Universal Robots PolyScope program: cube_dev.urp

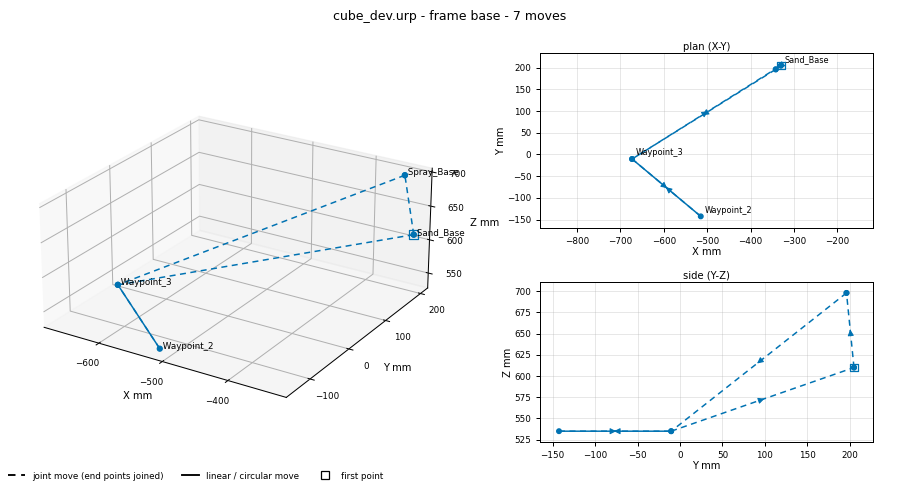
[picture p0: tool path of cube_dev.urp in frame base, 7 of 7 moves have a stored position in this frame; points joined in program order, loops and branches not executed]
Program cube_dev (installation=default directory=/programs/cube createdIn=5.11.5.1010327 lastSavedIn=5.11.5.1010327 robotSerialNumber=20215500677)
Calibrated DH parameters: a=[0.000204, -0.239222, -0.391845, -0.000001, 0.000022, 0]; d=[0.162722, -355.808559, 353.37206, 2.570385, 0.099741, 0.099629]; alpha=[1.571124, 0.000988, 0.008295, 1.568963, -1.570303, 0]; deltaTheta=[0, -0.973091, 7.204745, 0.05153, 0, 0]
Robot Program (runOnlyOnce=true)
  MoveJ speed 120 deg/s, acceleration 120 deg/s^2 (useActiveTCP=false) tcp=SandTCP; feature=Point_1
    Waypoint Sand_Base: TCP in base x=-330.026 y=205.009 z=609.986 mm, rx=0.0001 ry=-0.0003 rz=-2.2419 rad; joints [-54.6, -77.456, 120.707, 90.609, -79.088, -168.284] deg; TCP offset x=1.003 y=125.541 z=104.154 mm, rx=-0.7854 ry=0 rz=0 rad; feature pose in base x=-330 y=205 z=610 mm, rx=0 ry=0 rz=-1.5843 rad
  Folder Sand
    MoveL speed 50 mm/s, acceleration 1200 mm/s^2 (useActiveTCP=false) tcp=SandTCP; feature=Base
      MoveDirectionNode (selectedDirection=ZPlus)
        Until TOOL_CONTACT_DETECTION (allowActions=false retraction=0.001 decelerationAcceleration=3 decelerationAngularAcceleration=34.906585)
      URCap Finishing Tool Control (Robotiq_Copilot, Robotiq Inc.) dataModel(ToolOutputNameKey=SanderOn, HackTriggeringContributionIsDefinedMethodKey=true)
    MoveL speed 50 mm/s, acceleration 1200 mm/s^2 (useActiveTCP=true) feature=Base
      Force Simple feature=Base; selection=[0, 0, 1, 0, 0, 0]; wrench=[0, 0, 5, 0, 0, 0]; limitsForce=[0.15, 0.15, 0.15, 1.047198, 1.047198, 1.047198]; limitsMotion=[0.1, 0.1, 0.1, 0.349066, 0.349066, 0.349066]
        MoveDirectionNode (selectedDirection=XMinus)
          Until DISTANCE (allowActions=false deceleration=3 distanceNodeType=BLEND) Distance=0.355; motionParameters(blendRadius=0.025)
        MoveDirectionNode (selectedDirection=YMinus)
          Until DISTANCE (allowActions=false deceleration=3 distanceNodeType=BLEND) Distance=0.355; motionParameters(blendRadius=0.025)
        MoveDirectionNode (selectedDirection=XPlus)
          Until DISTANCE (allowActions=false deceleration=3 distanceNodeType=BLEND) Distance=0.355; motionParameters(blendRadius=0.025)
        MoveDirectionNode (selectedDirection=YPlus)
          Until DISTANCE (allowActions=false deceleration=3 distanceNodeType=STOP) Distance=0.355; motionParameters(blendRadius=0.01)
        URCap Finishing Tool Control (Robotiq_Copilot, Robotiq Inc.) dataModel(FinishingToolStateKey=false, ToolOutputNameKey=SanderOn, HackTriggeringContributionIsDefinedMethodKey=true)
    MoveL speed 90 mm/s, acceleration 1200 mm/s^2 (useActiveTCP=false) tcp=SandTCP; feature=Base
      MoveDirectionNode (selectedDirection=ZMinus)
        Until DISTANCE (allowActions=false deceleration=3 distanceNodeType=BLEND) Distance=0.05; motionParameters(blendRadius=0.003)
  Folder Spray Vert
    MoveJ speed 120 deg/s, acceleration 150 deg/s^2 (useActiveTCP=false) tcp=SprayTCP; feature=Point_1
      Waypoint Spray_Base: TCP in base x=-341.952 y=196.173 z=697.866 mm, rx=0 ry=0 rz=0.0032 rad; joints [-64.094, -80.171, 99.151, 94.355, -50.864, 55.964] deg; TCP offset x=-61.38 y=-97.07 z=93.78 mm, rx=0.6139 ry=0.6139 rz=-1.4822 rad; feature pose in base x=-341.965 y=196.202 z=697.85 mm, rx=0 ry=0 rz=-1.5843 rad
    MoveL speed 90 mm/s, acceleration 1200 mm/s^2 (useActiveTCP=false) tcp=SprayTCP; feature=Base
      MoveDirectionNode (selectedDirection=ZMinus)
        Until DISTANCE (allowActions=false deceleration=3 distanceNodeType=BLEND) Distance=0.05; motionParameters(blendRadius=0.003)
      Set DigitalOutput pin=SprayerOn; digitalValue=1
      MoveDirectionNode (selectedDirection=XMinus)
        Until DISTANCE (allowActions=false deceleration=3 distanceNodeType=BLEND) Distance=0.355; motionParameters(blendRadius=0.003)
      MoveDirectionNode (selectedDirection=YMinus)
        Until DISTANCE (allowActions=false deceleration=3 distanceNodeType=BLEND) Distance=0.355; motionParameters(blendRadius=0.003)
      MoveDirectionNode (selectedDirection=XPlus)
        Until DISTANCE (allowActions=false deceleration=3 distanceNodeType=BLEND) Distance=0.355; motionParameters(blendRadius=0.003)
      MoveDirectionNode (selectedDirection=YPlus)
        Until DISTANCE (allowActions=false deceleration=3 distanceNodeType=BLEND) Distance=0.355; motionParameters(blendRadius=0.003)
      Set DigitalOutput pin=SprayerOn; digitalValue=0
  Folder Spray Horiz
    MoveJ speed 120 deg/s, acceleration 150 deg/s^2 (useActiveTCP=false) tcp=SprayTCP; feature=Point_1
      Waypoint Spray_Base: TCP in base x=-341.952 y=196.173 z=697.866 mm, rx=0 ry=0 rz=0.0032 rad; joints [-64.094, -80.171, 99.151, 94.355, -50.864, 55.964] deg
      Waypoint Waypoint_3: TCP in base x=-672.939 y=-10.387 z=534.985 mm, rx=0.6191 ry=0.6108 rz=-1.4946 rad; joints [-18.021, -51.518, 72.974, -111.482, 90.452, 107.054] deg; TCP offset x=63.143 y=-107.882 z=84.395 mm, rx=0.6139 ry=0.6139 rz=-1.4822 rad; feature pose in base x=-330 y=205 z=580 mm, rx=0 ry=0 rz=-1.5843 rad
      Set DigitalOutput pin=SprayerOn; digitalValue=1
      MoveL speed 100 mm/s, acceleration 1200 mm/s^2 (useActiveTCP=false) tcp=SprayTCP; feature=Point_1
        MoveDirectionNode (selectedDirection=XPlus) feature=Base
          Until DISTANCE (allowActions=false deceleration=3 distanceNodeType=STOP) Distance=0.34; motionParameters(blendRadius=0)
        Set DigitalOutput pin=SprayerOn; digitalValue=0
        Waypoint Waypoint_2: motionParameters(jointSpeed=1.047198 jointAcceleration=1.396263 cartesianSpeed=0.25 cartesianAcceleration=1.2); TCP in base x=-514.712 y=-142.523 z=534.993 mm, rx=0.006 ry=0.8727 rz=-0.0126 rad; joints [6.181, -60.479, 87.661, -122.171, 89.804, 172.784] deg; TCP offset x=63.143 y=-107.882 z=84.395 mm, rx=0.6139 ry=0.6139 rz=-1.4822 rad
        Set DigitalOutput pin=SprayerOn; digitalValue=1
        MoveDirectionNode (selectedDirection=YPlus) feature=Base
          Until DISTANCE (allowActions=false deceleration=3 distanceNodeType=STOP) Distance=0.34; motionParameters(blendRadius=0)
        Set DigitalOutput pin=SprayerOn; digitalValue=0
      MoveJ speed 120 deg/s, acceleration 150 deg/s^2 (useActiveTCP=false) tcp=SprayTCP; feature=Point_1
        Waypoint Waypoint_1: TCP in base x=-672.939 y=-10.387 z=534.983 mm, rx=-0.7421 ry=0.7525 rz=1.4257 rad; joints [1.444, -66.75, 94.166, -117.891, 100.412, -92.529] deg; TCP offset x=63.143 y=-107.882 z=84.395 mm, rx=0.6139 ry=0.6139 rz=-1.4822 rad
        Set DigitalOutput pin=SprayerOn; digitalValue=1
      MoveL speed 100 mm/s, acceleration 1200 mm/s^2 (useActiveTCP=true) feature=Base
        MoveDirectionNode (selectedDirection=XPlus) feature=Base
          Until DISTANCE (allowActions=false deceleration=3 distanceNodeType=STOP) Distance=0.34; motionParameters(blendRadius=0)
        Set DigitalOutput pin=SprayerOn; digitalValue=0
  MoveJ speed 120 deg/s, acceleration 120 deg/s^2 (useActiveTCP=false) tcp=SandTCP; feature=Point_1
    Waypoint Sand_Base: TCP in base x=-330.026 y=205.009 z=609.986 mm, rx=0.0001 ry=-0.0003 rz=-2.2419 rad; joints [-54.6, -77.456, 120.707, 90.609, -79.088, -168.284] deg; TCP offset x=1.003 y=125.541 z=104.154 mm, rx=-0.7854 ry=0 rz=0 rad; feature pose in base x=-330 y=205 z=610 mm, rx=0 ry=0 rz=-1.5843 rad
